TYPE ST_RecipeStep :
STRUCT
	eCommand 	: E_RecipeStepCommand;
	fTarget 	: LREAL;
	tDuration	: TIME;
END_STRUCT
END_TYPE

(* stored: Version 1.1.0.1, ProductVersion 3.1.4024.15
   DUT ST_RecipeStep: Id {6d099065-c926-4c66-b30b-290277840c9c} *)
